// Mitsubishi GX Works2 project: pr3   PLC: Q03UDV

PROGRAM MAIN
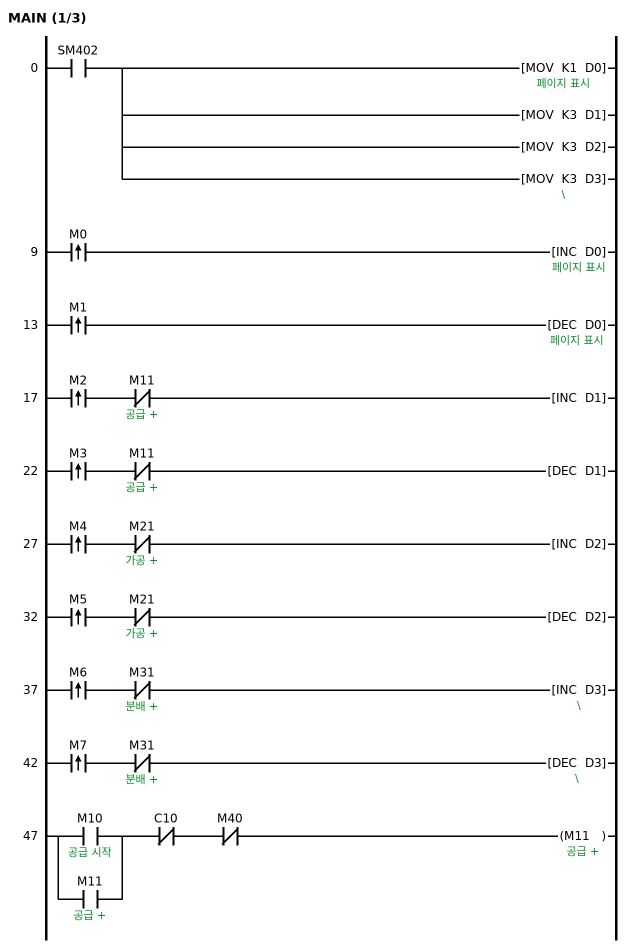
0     LD      SM402
      MOV     K1 D0  ; 페이지 표시
      MOV     K3 D1
      MOV     K3 D2
      MOV     K3 D3  ; \
9     LDP     M0
      INC     D0
13    LDP     M1
      DEC     D0
17    LDP     M2
      ANI     M11  ; 공급 +
      INC     D1
22    LDP     M3
      ANI     M11  ; 공급 +
      DEC     D1
27    LDP     M4
      ANI     M21  ; 가공 +
      INC     D2
32    LDP     M5
      ANI     M21  ; 가공 +
      DEC     D2
37    LDP     M6
      ANI     M31  ; 분배 +
      INC     D3
42    LDP     M7
      ANI     M31  ; 분배 +
      DEC     D3
47    LD      M10  ; 공급 시작
      OR      M11  ; 공급 +
      ANI     C10
      ANI     M40
      OUT     M11  ; 공급 +
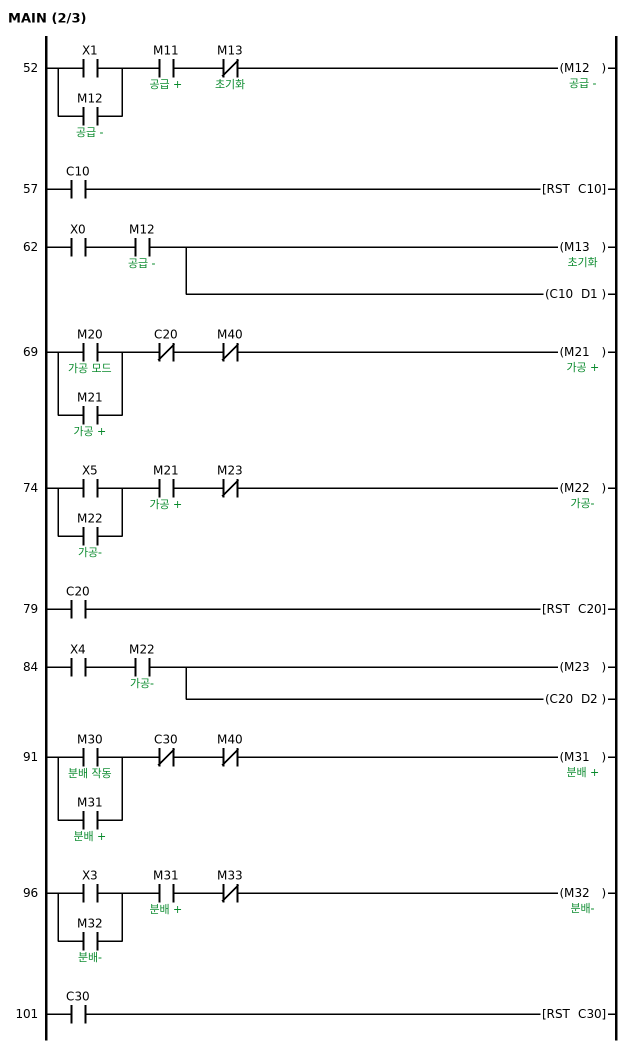
52    LD      X1
      OR      M12  ; 공급 -
      AND     M11  ; 공급 +
      ANI     M13  ; 초기화
      OUT     M12  ; 공급 -
57    LD      C10
      RST     C10
62    LD      X0
      AND     M12  ; 공급 -
      OUT     M13  ; 초기화
      OUT     C10 D1
69    LD      M20  ; 가공 모드
      OR      M21  ; 가공 +
      ANI     C20
      ANI     M40
      OUT     M21  ; 가공 +
74    LD      X5
      OR      M22  ; 가공-
      AND     M21  ; 가공 +
      ANI     M23
      OUT     M22  ; 가공-
79    LD      C20
      RST     C20
84    LD      X4
      AND     M22  ; 가공-
      OUT     M23
      OUT     C20 D2
91    LD      M30  ; 분배 작동
      OR      M31  ; 분배 +
      ANI     C30
      ANI     M40
      OUT     M31  ; 분배 +
96    LD      X3
      OR      M32  ; 분배-
      AND     M31  ; 분배 +
      ANI     M33
      OUT     M32  ; 분배-
101   LD      C30
      RST     C30
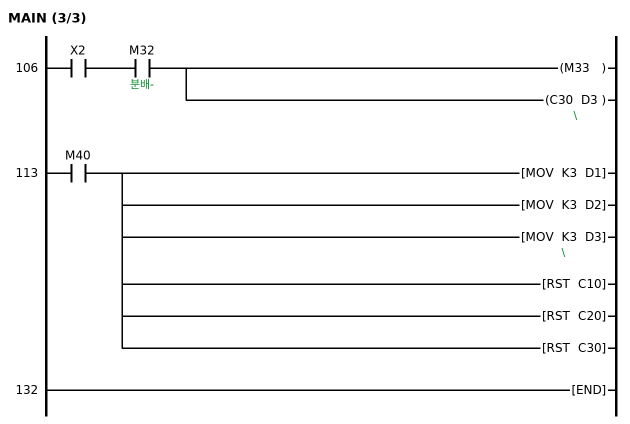
106   LD      X2
      AND     M32  ; 분배-
      OUT     M33
      OUT     C30 D3  ; \
113   LD      M40
      MOV     K3 D1
      MOV     K3 D2
      MOV     K3 D3
      RST     C10
      RST     C20
      RST     C30
132   END
END_PROGRAM

PROGRAM OUTPUT
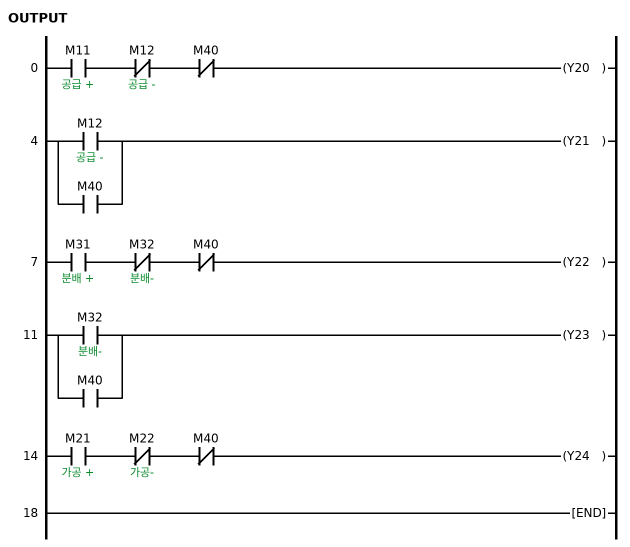
0     LD      M11  ; 공급 +
      ANI     M12  ; 공급 -
      ANI     M40
      OUT     Y20
4     LD      M12  ; 공급 -
      OR      M40
      OUT     Y21
7     LD      M31  ; 분배 +
      ANI     M32  ; 분배-
      ANI     M40
      OUT     Y22
11    LD      M32  ; 분배-
      OR      M40
      OUT     Y23
14    LD      M21  ; 가공 +
      ANI     M22  ; 가공-
      ANI     M40
      OUT     Y24
18    END
END_PROGRAM

// device comments not shown above
X15  ; 회전
X16  ; 회전 정지
X20  ; 가 모 버
X21  ; 컨 모 버
X22  ; 공 전 버
X30  ; 컨 모 버
X40  ; 공 전 버
X41  ; 공 후 버
Y0D  ; 드릴
Y2D  ; 드릴
Y2E  ; 컨베이어
